(*
Stores raw I_Component value and additional metadata.
*)
INTERFACE I_Component EXTENDS I_ComponentNode

(*
Returns parent Entity.
*)
PROPERTY Entity : I_Entity
GET
END_GET
END_PROPERTY

(*
Returns raw I_Component pointer.
*)
PROPERTY Raw : I_RawComponent
GET
END_GET
END_PROPERTY

END_INTERFACE

(* stored: Version 1.1.0.1
   Itf I_Component: Id {9272b1ca-5046-44a6-8849-d09e16589182}
   Property Entity: Id {d4c35409-a76d-443d-9b90-a15760e51851}
   Get Get: Id {3588b483-3719-4cdd-b6a9-8f7e565c8021}
   Property Raw: Id {7d416757-8acb-4146-ae12-90b882db77a8}
   Get Get: Id {e25140a9-a228-42c9-9678-c44e1c0faa3c} *)
